// TwinCAT 3 PLC project Main
// ProgramVersion: 3.1.4024.0
// libraries:
//   Tc2_Standard, * (Beckhoff Automation GmbH)
//   Tc2_System, * (Beckhoff Automation GmbH)
//   Tc3_Module, * (Beckhoff Automation GmbH)
//   Tc3_Vision, * (Beckhoff Automation GmbH)
//   TcUnit, * (www.tcunit.org)
// project tree:
//   / PlcTask.TcTTO
//   POUs/Library/Animation/ SpriteSheetAnimationFrames.TcPOU
//   POUs/Library/EL2574/ EL2574_ExtendedMode.TcPOU (not stored)
//   POUs/Library/ImageSerializer/Base/ ImageSerializer.TcPOU (not stored)
//   POUs/Library/ImageSerializer/Interfaces/ I_ImageSerializer.TcIO (not stored)
//   POUs/Library/ImageSerializer/Matrix/ MatrixImageSerializer.TcPOU
//   POUs/Library/ImageSerializer/Null/ NullImageSerializer.TcPOU (not stored)
//   POUs/Library/PixelReader/ I_PixelReader.TcIO (not stored), EL2574PixelReader.TcPOU (not stored)
//   POUs/ MAIN.TcPOU
//   Tests/ EL2574PixelReader_TestSuite.TcPOU (not stored), UnitTests.TcPOU (not stored)
// real-time tasks:
//   TASK PlcTask: cycle T#200us, priority 20, ADS port 350
// I/O:
//   DEVICE Device 3 (EtherCAT)
// variable links:
//   Main Instance <-> Device 3 (EtherCAT)/Term 1 (EK1100)/Term 4 (EL2574)
//     PlcTask Inputs/MAIN.el2574.pdo.MDP5001_260_Input/MDP5001_260_Status <-> SlotGroup 1 (Slot 1, 2) (1xASYNC)/Status Channel 1/Status
//     PlcTask Outputs/MAIN.el2574.pdo.MDP5001_260_Output/MDP5001_260_Extended_Control <-> SlotGroup 1 (Slot 1, 2) (1xASYNC)/Extended Channel 1/Extended Control

CONFIGURATION Main
    RESOURCE PLC ON TwinCAT3
        TASK PlcTask(INTERVAL := T#200us, PRIORITY := 20);
        PROGRAM MAIN WITH PlcTask : MAIN;
    END_RESOURCE
END_CONFIGURATION

// ---- POUs/MAIN.TcPOU
PROGRAM MAIN
VAR
	// demo triggers
	startAnimation : BOOL := TRUE;
	clear : BOOL := FALSE;
	
	// helpers
	animation : SpriteSheetAnimationFrames(
		SpriteSheetFilePath := 'C:\temp\christmas-invert.png',
		SpriteWidth := 32,
		SpriteHeight := 16,
		TotalSprites := 46,
		Columns := 2,
		Rows := 3
	);

	// equipment
	matrix1 : MatrixImageSerializer(Height := 16, Width := 16, X := 0, Y := 0); // 0 - 255
	matrix2 : MatrixImageSerializer(Height := 16, Width := 16, X := 16, Y := 0); // 256 - 511
	el2574 : EL2574_ExtendedMode(TotalPixels := 512); // you need to pass in the total number of pixels connected to the EK2574
	
	// program variables
	initialized : BOOL;
	animationRTrigger : R_TRIG;
	animationTimer : ton;
	
END_VAR

(*

  _____ __  __ _____   ____  _____ _______       _   _ _______ _ 
 |_   _|  \/  |  __ \ / __ \|  __ \__   __|/\   | \ | |__   __| |
   | | | \  / | |__) | |  | | |__) | | |  /  \  |  \| |  | |  | |
   | | | |\/| |  ___/| |  | |  _  /  | | / /\ \ | . ` |  | |  | |
  _| |_| |  | | |    | |__| | | \ \  | |/ ____ \| |\  |  | |  |_|
 |_____|_|  |_|_|     \____/|_|  \_\ |_/_/    \_\_| \_|  |_|  (_)
 
Competition Clause: 

During the Beckhoff Christmas coding competition involving the EL2574 
LED controller terminal, if any Beckhoff subsidiaries use, borrow from, or are inspired
by this code for their own competition entry, they must acknowledge the inspiration by 
including the hashtag #codingbytes in any LinkedIn posts related to their competition entry. 
This requirement is in effect until the conclusion OF the competition on 25th December 2024.

*)

IF NOT initialized THEN
	// First setup the wiring of the units.  This must be in the order they are physically connected.
	matrix1.ConnectTo(matrix2);
	// that's initializing done!
	initialized := TRUE;
END_IF

// we wait here until the animation source image is loaded.
// i.e. we return, which prevents the program from progressing past this line.
IF NOT animation.TryLoad() THEN
    RETURN;
END_IF

// basic clear trigger.  Set clear TRUE to clear the display
IF clear AND_THEN el2574.TrySendClearAll() THEN
	clear := FALSE;
END_IF

// animation logic.  Set startAnimation to TRUE to begin the animation.

// just to make things tidy, when a rising edge is detected on startAnimation then
// reset the animation to the start.
animationRTrigger(Clk:=startAnimation);
IF animationRTrigger.Q THEN
	animation.MoveToStart();
END_IF

// using a simple pulsing timer of 100ms, update the image in the connected matrixs and 
// tell the terminal to display the new frame.
//
// if we can no longer move to the next frame, then this means we are at the end, so 
// we tell the animation to start again. 
animationTimer(in:=NOT animationTimer.q, pt:=T#100MS);
IF startAnimation AND animationTimer.Q THEN
		
	matrix1.UpdateImage(animation.CurrentFrameImage);
	el2574.TrySendPixelsFromSerializer(matrix1);
	
	IF NOT animation.TryMoveNext() THEN
		animation.MoveToStart();
	END_IF

END_IF

// cyclic call the terminal so that it can do it's job.
el2574.CyclicCall();

// unit tests
UnitTests();

END_PROGRAM

// ---- POUs/Library/Animation/SpriteSheetAnimationFrames.TcPOU
FUNCTION_BLOCK SpriteSheetAnimationFrames
VAR
	spriteSheetFilePath : T_MAXSTRING;
	spriteWidth : UDINT;
	spriteHeight : UDINT;
	totalSprites : UDINT;
	columns : UDINT;
	rows : UDINT;
	spriteSheetImage : ITcVnImage;
	readImage: FB_VN_ReadImage;
	
	// animation variables
	_currentFrameIndex : UDINT;
	_currentFrameImage : ITcVnImage;
END_VAR

PROPERTY PUBLIC CurrentFrameImage : ITcVnImage
GET
CurrentFrameImage := _currentFrameImage;
END_GET
END_PROPERTY

PROPERTY PUBLIC CurrentFrameIndex : UDINT
GET
CurrentFrameIndex := _currentFrameIndex;
END_GET
END_PROPERTY

METHOD FB_init : BOOL
VAR_INPUT
	bInitRetains : BOOL; // if TRUE, the retain variables are initialized (warm start / cold start)
	bInCopyCode : BOOL;  // if TRUE, the instance afterwards gets moved into the copy code (online change)
	SpriteSheetFilePath : T_MAXSTRING;
	SpriteWidth : UDINT;
	SpriteHeight : UDINT;
	TotalSprites : UDINT;
	Columns : UDINT;
	Rows : UDINT;
END_VAR
THIS^.spriteSheetFilePath := SpriteSheetFilePath;
THIS^.spriteWidth := SpriteWidth;
THIS^.spriteHeight := SpriteHeight;
THIS^.totalSprites := TotalSprites;
THIS^.columns := Columns;
THIS^.rows := Rows;
END_METHOD

PROPERTY PUBLIC IsAtLastFrame : BOOL
GET
IF TotalFrameCount = 0 THEN
	IsAtLastFrame := TRUE;
	RETURN;
END_IF

IsAtLastFrame := CurrentFrameIndex = TotalFrameCount - 1;
END_GET
END_PROPERTY

METHOD PUBLIC MoveToStart
VAR_INPUT
END_VAR
_currentFrameIndex := 0;
TryGetSprite(_currentFrameIndex, _currentFrameImage);
END_METHOD

PROPERTY PUBLIC TotalFrameCount : UDINT
GET
TotalFrameCount := totalSprites;
END_GET
END_PROPERTY

METHOD PRIVATE TryGetSprite : BOOL
VAR_INPUT
	Index : UDINT;
	Destination : REFERENCE TO ITcVnImage;
END_VAR
VAR
	spriteX : UDINT;
	spriteY : UDINT;
	spriteColumn : UDINT;
	spriteRow : UDINT;
	result : HRESULT;
END_VAR
IF Index > TotalFrameCount - 1 THEN
	RETURN;
END_IF

spriteColumn := Index MOD columns;
spriteRow := Index / columns;

spriteX := spriteColumn * spriteWidth;
spriteY := spriteRow * spriteHeight;

result := F_VN_CopyImage(spriteSheetImage, _currentFrameImage, s_OK);
result := F_VN_SetRoi(spriteX, spriteY, spriteWidth, spriteHeight, _currentFrameImage, result);

TryGetSprite := Succeeded(result);
END_METHOD

METHOD PUBLIC TryLoad : BOOL
VAR
	i : UDINT;
END_VAR
// if we already have an image loaded, then we can early jump out as we know everything is done. 
IF spriteSheetImage <> 0 THEN
	TryLoad := TRUE;
	RETURN;
END_IF

IF spriteSheetFilePath = '' OR  spriteWidth = 0 OR spriteHeight = 0 OR totalSprites = 0 OR columns = 0 OR rows = 0 THEN
	// this is our sanity check, we return out if anything is bad.
	// if we pass this point we know we can use the variables confidently.
	RETURN;
END_IF

// we keep polling the read until an image is read.  If it faults due to error then we just sit here and never return true.
readImage(sFilePath := spriteSheetFilePath, ipDestImage := spriteSheetImage, bRead := TRUE, nTimeout := T#500MS);
IF readImage.bBusy THEN 
	RETURN;
END_IF

IF readImage.bError THEN 
	RETURN;
END_IF 

// at this point we should have an image, so we will do one final check before moving on.  
IF spriteSheetImage = 0 THEN
	RETURN;
END_IF

// we have made it this far, which means we need to set the CurrentFrameImage to the first part of the image and report as done. 
MoveToStart();
TryLoad := TRUE;
END_METHOD

METHOD PUBLIC TryMoveNext : BOOL
VAR_INPUT
END_VAR
IF _currentFrameIndex = TotalFrameCount - 1 THEN
	RETURN;
END_IF

_currentFrameIndex := _currentFrameIndex + 1;
TryMoveNext := TryGetSprite(_currentFrameIndex, _currentFrameImage);
END_METHOD

END_FUNCTION_BLOCK

// ---- POUs/Library/ImageSerializer/Matrix/MatrixImageSerializer.TcPOU
FUNCTION_BLOCK MatrixImageSerializer EXTENDS ImageSerializer
VAR
	height : UDINT;
	width : UDINT;
	x : UDINT;
	y : UDINT;
	image : ITcVnImage;
	live : ITcVnDisplayableImage; // used in this demo to show the image for the matrix
	_pixelCount : UDINT;
END_VAR

METHOD FB_init : BOOL
VAR_INPUT
	bInitRetains : BOOL; // if TRUE, the retain variables are initialized (warm start / cold start)
	bInCopyCode : BOOL;  // if TRUE, the instance afterwards gets moved into the copy code (online change)
	Height : UDINT;
	Width : UDINT;
	X : UDINT;
	Y : UDINT;
END_VAR
THIS^.height := Height;
THIS^.width := Width;
THIS^.x := X;
THIS^.y := Y;

Initialize();
END_METHOD

METHOD PRIVATE Initialize
VAR_INPUT
END_VAR
_pixelCount := width * height;
END_METHOD

METHOD PROTECTED OnTryGetPixel : BOOL
VAR_INPUT
	PixelIndex : UDINT;
	Reader : I_PixelReader;
END_VAR
VAR
	xPosition : UDINT;
	yPosition : UDINT;
END_VAR
IF width = 0 OR height = 0 THEN
	RETURN;
END_IF

xPosition := PixelIndex MOD width;
yPosition := PixelIndex / width;

// If it's an odd row, reverse the direction
IF yPosition MOD 2 = 1 THEN 
    xPosition := (width - 1) - xPosition;
END_IF

OnTryGetPixel := succeeded(F_VN_GetPixel(image, Reader.Value, xPosition, yPosition, s_OK));
END_METHOD

METHOD PROTECTED OnUpdateImage
VAR_INPUT
	Source : ITcVnImage;
END_VAR
VAR
	result : HRESULT;
END_VAR
result := F_VN_CopyImage(Source, image, s_OK);
result := F_VN_SetRoi(x, y, width, height, image, result);

IF Succeeded(result) THEN
	F_VN_CopyIntoDisplayableImage(image, live, s_ok);
	RETURN;
END_IF

// there was an error, so best to clear the internal image as it's no longer valid.
// but only if there was an image there in fht first place.

IF image = 0 THEN
	RETURN;
END_IF

image.TcRelease();
image := 0;
END_METHOD

{attribute 'monitoring' := 'call'}
PROPERTY PUBLIC PixelCount : UDINT
GET
PixelCount := _pixelCount;
END_GET
END_PROPERTY

END_FUNCTION_BLOCK
